(* IEC 61131-3 sources: DatObjWrap/, 4 files *)

(* ---- DatObjWrap.typ ---- *)
(********************************************************************
 * COPYRIGHT -- B&R Industrial Automation
 ********************************************************************
 * Library: DatObjWrap
 * File: DatObjWrap.typ
 * Author: blackburnd
 * Created: March 10, 2010
 ********************************************************************
 * Data types of library DatObjWrap
 ********************************************************************)

TYPE
	DOWRAP_OP_enum :
		(
		DOWRAP_OP_INVALID := 0,
		DOWRAP_OP_OPEN,
		DOWRAP_OP_SAVEAS
		);
	DOWRAP_ST_enum :
		(
		DOWRAP_ST_WAIT := 0, (*0*)
		DOWRAP_ST_GETINFO, (*1*)
		DOWRAP_ST_CREATE, (*2*)
		DOWRAP_ST_OPEN, (*3*)
		DOWRAP_ST_SAVE, (*4*)
		DOWRAP_ST_ERROR := 999, (*999*)
		DOWRAP_ST_
		);
	DatObjWrap_Int_FUB_typ : 	STRUCT
		DatObjGetInfo : DatObjInfo;
		DatObjCreate : DatObjCreate;
		DatObjWrite : DatObjWrite;
		DatObjRead : DatObjRead;
	END_STRUCT;
	DatObjWrap_Internal_typ : 	STRUCT
		Ident : UDINT; (*Data object ident*)
		State : DINT; (*State variable*)
		CurrOperation : DINT; (*Current operation (Save or Load)*)
		FUB : DatObjWrap_Int_FUB_typ;
		CMD : DatObjWrap_IN_CMD_typ;
	END_STRUCT;
	DatObjWrap_OUT_STAT_typ : 	STRUCT
		Busy : BOOL; (*Object is busy performing an action*)
		Done : BOOL; (*Action finished successfully*)
		Error : BOOL; (*There is an error with the DOHandling*)
		ErrorID : UINT; (*Error number from internal FUBs*)
		ErrorString : STRING[DOWRAP_STRLEN_ERROR];
		ErrorLevel : USINT;
		ErrorState : DINT; (*State in which error occurred*)
	END_STRUCT;
	DatObjWrap_OUT_typ : 	STRUCT
		STAT : DatObjWrap_OUT_STAT_typ;
	END_STRUCT;
	DatObjWrap_IN_PAR_typ : 	STRUCT
		DataObjName : STRING[8]; (*Name of the data object to which to store data*)
		pData : UDINT; (*Pointer to the data location to be saved from/loaded to*)
		len : UDINT; (*Length of the data to be saved/loaded*)
	END_STRUCT;
	DatObjWrap_IN_CMD_typ : 	STRUCT
		Open : BOOL; (*Load settings from Data Object.*)
		SaveAs : BOOL; (*Save settings to Data Object.*)
		AcknowledgeError : BOOL; (*Acknowledge errors*)
	END_STRUCT;
	DatObjWrap_IN_typ : 	STRUCT
		CMD : DatObjWrap_IN_CMD_typ;
		PAR : DatObjWrap_IN_PAR_typ;
	END_STRUCT;
	DatObjWrap_typ : 	STRUCT
		IN : DatObjWrap_IN_typ;
		OUT : DatObjWrap_OUT_typ;
		Internal : DatObjWrap_Internal_typ;
	END_STRUCT;
END_TYPE

(* ---- DatObjWrap.fun ---- *)
(********************************************************************
 * COPYRIGHT -- B&R Industrial Automation
 ********************************************************************
 * Library: DatObjWrap
 * File: DatObjWrap.fun
 * Author: blackburnd
 * Created: March 10, 2010
 ********************************************************************
 * Functions and function blocks of library DatObjWrap
 ********************************************************************)

FUNCTION DatObjWrapFn_Cyclic : BOOL (*This function implements a wrapper for Data Object writing and reading.*)
	VAR_IN_OUT
		t : DatObjWrap_typ; (*Data object wrapper control object.*)
	END_VAR
END_FUNCTION

FUNCTION DatObjWrapOpen_Init : BOOL (*Synchronously loads a data object. Should ONLY be called in the INIT routine.*)
	VAR_IN_OUT
		t : DatObjWrap_typ; (*Data object wrapper control object.*)
	END_VAR
END_FUNCTION

FUNCTION dowSetError : BOOL (*Set error status on DatObjWrap*)
	VAR_INPUT
		ErrorID : UINT;
	END_VAR
	VAR_IN_OUT
		t : DatObjWrap_typ;
	END_VAR
END_FUNCTION

(* ---- dowSetError.st ---- *)
(********************************************************************
 * COPYRIGHT -- Automation Resources Group
 ********************************************************************
 * Library: DatObjWrap
 * File: dowSetError.st
 * Author: David Blackburn
 * Created: December 22, 2011
 ********************************************************************
 * Implementation of library DatObjWrap
 ********************************************************************)

(********************************************************************)
(* Set error status on DatObjWrap 									*)
(********************************************************************)

(* Reset Busy, Done			DONE and TESTED DFB 20111222 *)
(* Set Error				DONE and TESTED DFB 20111222 *)
(* Set ErrorID				DONE and TESTED DFB 20111222 *)
(* Set ErrorLevel			DONE and TESTED DFB 20111222 *)
(* Set ErrorState			DONE and TESTED DFB 20111222 *)
(* Set State				DONE and TESTED DFB 20111222 *)
(* Set ErrorString			DONE and TESTED DFB 20111222 *)

FUNCTION dowSetError

(****************************************************)
(* Set return value to get rid of compile warning 	*)
(****************************************************)

dowSetError:=	FALSE;

(************************************************)
(* Set error status								*)
(************************************************)

t.OUT.STAT.Busy:=		0;
t.OUT.STAT.Done:=		0;
t.OUT.STAT.Error:=		1;
t.OUT.STAT.ErrorID:=	ErrorID;
t.OUT.STAT.ErrorLevel:=	3;
t.OUT.STAT.ErrorState:=	t.Internal.State;
t.Internal.State:=		DOWRAP_ST_ERROR;

(* Set ErrorString *)

CASE ErrorID OF

	0: t.OUT.STAT.ErrorString:=	'';

	doERR_ILLPARAMETER:			t.OUT.STAT.ErrorString:=	'Invalid parameter. Check IN.PAR.pData.';
	doERR_DUPOBJECT:			t.OUT.STAT.ErrorString:=	'Object already present.';
	doERR_ILLMEMTYPE:			t.OUT.STAT.ErrorString:=	'Invalid memory type.';
	doERR_NOMEMORY:				t.OUT.STAT.ErrorString:=	'No memory available for object.';
	doERR_BRINSTALL:			t.OUT.STAT.ErrorString:=	'Error installing data object.';
	doERR_ILLOBJECT:			t.OUT.STAT.ErrorString:=	'Data object not found. Check IN.PAR.DataObjName.';
	doERR_ILLOBJTYPE:			t.OUT.STAT.ErrorString:=	'Object found, but it was not a data object. Check IN.PAR.DataObjName.';
	doERR_WRONGOFFSET:			t.OUT.STAT.ErrorString:=	'Invalid offset specified.';
	doERR_ILLEGALLENGTH:		t.OUT.STAT.ErrorString:=	'Invalid length specified. Check IN.PAR.len.';
	doERR_MODULNOTFOUND:		t.OUT.STAT.ErrorString:=	'Data object not found. Check IN.PAR.DataObjName.';
	doERR_WRONGTIME:			t.OUT.STAT.ErrorString:=	'Invalid date set.';
	doERR_ILLSTATE:				t.OUT.STAT.ErrorString:=	'Data object not in correct state.';
	doERR_STARTHANDLER:			t.OUT.STAT.ErrorString:=	'System error.';
	doERR_TOOLONG_MODULNAME:	t.OUT.STAT.ErrorString:=	'Data object name is too long. Check IN.PAR.DataObjName.';
	doERR_BURNINGOBJECT:		t.OUT.STAT.ErrorString:=	'System error.';

	ELSE	t.OUT.STAT.ErrorString:=	'Unknown error.';

END_CASE

END_FUNCTION

(* ---- DatObjWrap.var ---- *)
(********************************************************************
 * COPYRIGHT -- B&R Industrial Automation
 ********************************************************************
 * Library: DatObjWrap
 * File: DatObjWrap.var
 * Author: blackburnd
 * Created: March 10, 2010
 ********************************************************************
 * Constants of library DatObjWrap
 ********************************************************************)
VAR CONSTANT
	DOWRAP_STATUS_FUB_DISABLED : UINT := 65534;
	DOWRAP_STRLEN_ERROR : USINT := 80;
END_VAR
